Staubli VAL3: iRack4.pgx

public program iRack4(num& nNum[] (dimensions=1))
begin
  nNum=dioGet(iRack4)
end
